Yaskawa INFORM job: JOBSTART.JBI

/JOB
//NAME JOBSTART
//POS
///NPOS 0,0,0,0,0,0
//INST
///DATE 2018/09/10 14:54
///ATTR SC,RW,MC
NOP
DOUT OG#(77) B001
DOUT OG#(78) B002
TIMER T=0.50
DOUT OT#(594) ON
TIMER T=0.50
DOUT OT#(595) OFF
TIMER T=0.50
END
